Yaskawa INFORM job: AAA.JBI

/JOB
//NAME AAA
//POS
///NPOS 0,0,1,0,0,0
///TOOL 12
///POSTYPE PULSE
///PULSE
EC00000=-29914,247808
//INST
///DATE 2025/09/01 15:32
///ATTR SC,RW
///GROUP1 ST1
NOP
MOVJ EC00000 VJ=40.0
END
